PROGRAM P_Init_einmalig
VAR
END_VAR

(* PU100 *)
GA_Global.Optimierer_Freigabe := 1;

END_PROGRAM

(* stored: Version 1.1.0.1, ProductVersion 3.1.4024.9
   POU P_Init_einmalig: Id {5f4fa04f-9f04-461b-9e7a-74e7253b8e41}, SpecialFunc None *)
